// Mitsubishi GX Works2 project: DE02   PLC: FX2N/FX2NC

PROGRAM MAIN
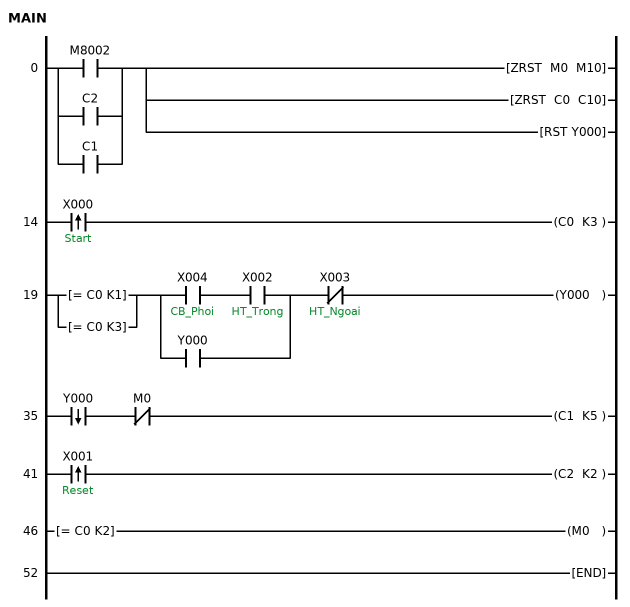
0     LD      M8002
      OR      C2
      OR      C1
      ZRST    M0 M10
      ZRST    C0 C10
      RST     Y000
14    LDP     X000  ; Start
      OUT     C0 K3
19    LD=     C0 K1
      OR=     C0 K3
      LD      X004  ; CB_Phoi
      AND     X002  ; HT_Trong
      OR      Y000
      ANB
      ANI     X003  ; HT_Ngoai
      OUT     Y000
35    LDF     Y000
      ANI     M0
      OUT     C1 K5
41    LDP     X001  ; Reset
      OUT     C2 K2
46    LD=     C0 K2
      OUT     M0
52    END
END_PROGRAM
